// TIA Portal V17 export
// export: Created 2022-12-08T07:31:26.4010087Z, ExportSetting WithDefaults, DisplayName Totally Integrated Automation Portal, DisplayVersion V17 Update 5, DisplayName TIA Portal Openness, DisplayVersion V17 Update 5, DisplayName TIA Portal Version Control Interface, DisplayVersion V17, DisplayName Simotion SCOUT TIA, DisplayVersion 5.4.3.0, DisplayName SINAMICS Startdrive Advanced, DisplayVersion V17 SP1, DisplayName SINAMICS Startdrive G130, G150, S120, S150, SINAMICS MV, S210, DisplayVersion V17 SP1, DisplayName SINAMICS Startdrive G110M, G120, G120C, G120D, G120P, G115D, DisplayVersion V17 SP1, DisplayName STEP 7 Professional, DisplayVersion V17 Update 5, DisplayName STEP 7 Safety, DisplayVersion V17, DisplayName WinCC Advanced, DisplayVersion V17 Update 5
DATA_BLOCK "DB_OperatingHour"   // DB105
AUTHOR : EconoPak GmbH
VERSION : 0.1
// stored: AutoNumber true, DBAccessibleFromOPCUA true, DBAccessibleFromWebserver true, InstanceOfName FB_OperatingHour, InstanceOfType FB
"FB_OperatingHour"
   // VAR_INPUT
   //    i_BtnReset : Bool;
   //    i_SafetyOk : Bool;
   //    i_Clock1Hz : Bool;
   // END_VAR
   // VAR_OUTPUT
   //    q_OperatingHoursList { ExternalAccessible := 'False'; ExternalVisible := 'False'; ExternalWritable := 'False'} : "UDT_OperatingHoursList";
   // END_VAR
   // VAR_IN_OUT
   //    iq_OMACGlobalData : "UDT_OMAC_GlobalData";
   // END_VAR
   // VAR
   //    inst_OperationCounter : Array[0..6] of "FB_OperatingHoursCounter";
   // END_VAR
BEGIN
END_DATA_BLOCK
